// TIA Portal V20 export
DATA_BLOCK "HMI_Test_DB"   // DB46
// stored: InstanceOfName HMI_Test, InstanceOfType FB
"HMI_Test"
   // VAR
   //    Old_Value : USInt;
   //    HMI_Connection_Alarm : Bool;
   //    Timer_2s : TON_TIME;
   // END_VAR
BEGIN
END_DATA_BLOCK
